(* PLC project Tc2_IoFunctions.IOF_GetDeviceName Demo, tc3-libraries-kb TwinCAT 3.1 *)
(* stored: creationDateTime 2026-05-21T00:00:00, modificationDateTime 2026-05-21T00:00:00 *)

PROGRAM P_Demo_IOF_GetDeviceName
  VAR
    fbGetDeviceName : IOF_GetDeviceName;  (* ID → 名字 FB *)
    sTargetNetId : T_AmsNetId := '';  (* 本机 *)
    nLookupDeviceId : UDINT := 1;  (* 要查的 Device Id *)
    bStartGetName : BOOL := FALSE;  (* 上升沿触发 *)
    tGetNameTimeout : TIME := T#5S;  (* 超时 *)
    bGetNameBusy : BOOL;  (* 工作中 *)
    bGetNameError : BOOL;  (* 失败 *)
    nLastErrCode : UDINT;  (* 错误号 *)
    sDeviceNameOut : T_MaxString;  (* 设备名 *)
  END_VAR

// =============================================================================
// 场景：IO 巡检脚本枚举所有 Device Id 后，对每个 ID 调本 FB 拿名字写到日志。
// 价值：可读诊断日志。
// 验证：登录后 nLookupDeviceId := 1，在线写 bStartGetName := TRUE → 回 FALSE 后 sDeviceNameOut 显示 System Manager 命名。
// 验证步骤：
//   1. 右键 PLC 项目 → Import PLCopenXML → 选本文件
//   2. 引用 Tc2_IoFunctions（References → Add library）
//   3. 编译 → 登录 → 运行；按上方『验证』行的指示在线写值观察
// =============================================================================

fbGetDeviceName(
    NETID      := sTargetNetId,
    DEVICEID   := nLookupDeviceId,
    START      := bStartGetName,
    TMOUT      := tGetNameTimeout,
    BUSY       => bGetNameBusy,
    ERR        => bGetNameError,
    ERRID      => nLastErrCode,
    DEVICENAME => sDeviceNameOut
);
END_PROGRAM
